METHOD mCallTop : E_cmdState
VAR_INPUT
	I_bExecute		: BOOL;
END_VAR
// No command requested.
IF NOT I_bExecute 
	THEN
    mCallTop       := E_CmdState.Idle;
    RETURN;
END_IF

// Command cylinder to top.
// ToBottom=FALSE, ToTop=TRUE.
fbBottomOut.bBoolValue 		 := FALSE;
fbTopOut.bBoolValue    	   := TRUE;

// Wait until top sensor is active.
IF fbTopIn.bBoolValue 
	THEN
		mCallTop 			 := E_CmdState.Succeeded;
ELSE
    mCallTop 			 := E_CmdState.Busy;
END_IF
END_METHOD

END_FUNCTION_BLOCK

// ---- 1000 Maschine xxx/_Customer/VISUs/Visu_Customer.TcVIS
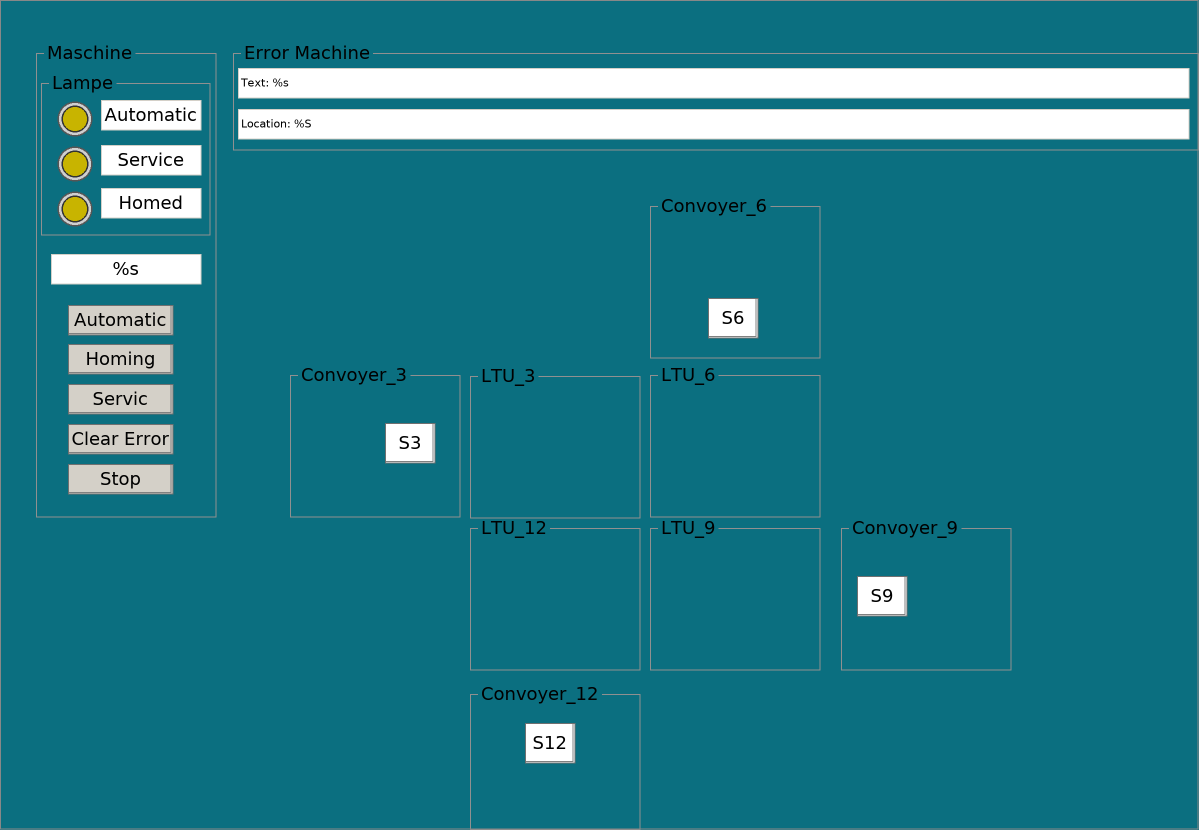
VISUALIZATION Visu_Customer  // 1199x830
    GroupBox (36,45 180x472), "Maschine"
        GroupBox (5,30 169x160), "Lampe"
            Lamp1 (14,114 40x40), variable: MAIN.fbCustomer.stHMI.bHomed, style: Lamp-Lamp1-Yellow
            Lamp1 (14,69 40x40), style: Lamp-Lamp1-Yellow
            Lamp1 (14,24 40x40), style: Lamp-Lamp1-Yellow
            Textfield (60,25 100x30), "Automatic"
            Textfield (60,70 100x30), "Service"
            Textfield (60,113 100x30), "Homed"
        Textfield (15,209 150x30), "%s", text variable: MAIN.fbCustomer.stHMI.eMode
            OnMouseClick: write the text variable via Default
        Button (32,419 105x30), "Stop"
        Button (32,379 105x30), "Clear Error"
        Button (32,339 105x30), "Servic", colour toggle: MAIN.fbCustomer.stHMI.bCmdService
            OnMouseClick: toggle MAIN.fbCustomer.stHMI.bCmdService
        Button (32,299 105x30), "Homing", colour toggle: MAIN.fbCustomer.stHMI.bCmdHome
            OnMouseClick: toggle MAIN.fbCustomer.stHMI.bCmdHome
        Button (32,260 105x30), "Automatic", text variable: MAIN.fbCustomer.stHMI.bCmdAuto, colour toggle: MAIN.fbCustomer.stHMI.bCmdAuto
            OnMouseClick: toggle MAIN.fbCustomer.stHMI.bCmdAuto
    GroupBox (290,367 170x150), "Convoyer_3"
        Button (95,56 50x40), "S3", colour toggle: MAIN.fbCustomer.fdConvoyerDevice3.fbStopperCarrieConvoyer.bHmiSimCarrie
            OnMouseClick: toggle MAIN.fbCustomer.fdConvoyerDevice3.fbStopperCarrieConvoyer.bHmiSimCarrie
    GroupBox (470,368 170x150), "LTU_3"
    GroupBox (650,367 170x150), "LTU_6"
    GroupBox (650,520 170x150), "LTU_9"
    GroupBox (470,520 170x150), "LTU_12"
    GroupBox (650,198 170x160), "Convoyer_6"
        Button (58,100 50x40), "S6", colour toggle: MAIN.fbCustomer.fdConvoyerDevice6.fbStopperCarrieConvoyer.bHmiSimCarrie
            OnMouseClick: toggle MAIN.fbCustomer.fdConvoyerDevice6.fbStopperCarrieConvoyer.bHmiSimCarrie
    GroupBox (470,686 170x144), "Convoyer_12"
        Button (55,37 50x40), "S12", colour toggle: MAIN.fbCustomer.fdConvoyerDevice12.fbStopperCarrieConvoyer.bHmiSimCarrie
            OnMouseClick: toggle MAIN.fbCustomer.fdConvoyerDevice12.fbStopperCarrieConvoyer.bHmiSimCarrie
    GroupBox (841,520 170x150), "Convoyer_9"
        Button (16,56 50x40), "S9", colour toggle: MAIN.fbCustomer.fdConvoyerDevice9.fbStopperCarrieConvoyer.bHmiSimCarrie
            OnMouseClick: toggle MAIN.fbCustomer.fdConvoyerDevice9.fbStopperCarrieConvoyer.bHmiSimCarrie
    GroupBox (233,45 966x105), "Error Machine"
        Textfield (5,23 951x30), "Text: %s"
        Textfield (5,64 951x30), "Location: %S"
END_VISUALIZATION

// ---- GlobalTextList.TcGTLO
TEXTLIST GlobalTextList
  325 = '%s'
  279 = '12'
  584 = 'Auto'
  173 = 'Automatic'
  1066 = 'BASEPOS'
  355 = 'BasePos'
  790 = 'C3'
  669 = 'C6'
  844 = 'Clear Error'
  626 = 'Convoyer_12'
  213 = 'Convoyer_3'
  419 = 'Convoyer_6'
  374 = 'Convoyer_9'
  648 = 'Error'
  908 = 'Error Machine'
  728 = 'Gruppenfeld'
  1008 = 'HOLD'
  917 = 'Homed'
  551 = 'Homing'
  218 = 'Lampe'
  354 = 'Location: %S'
  649 = 'LTU6'
  478 = 'Ltu_12'
  324 = 'LTU_12'
  891 = 'Ltu_3'
  699 = 'LTU_3'
  330 = 'Ltu_6'
  225 = 'LTU_6'
  558 = 'Ltu_9'
  195 = 'LTU_9'
  56 = 'Machine Desk'
  924 = 'Maschine'
  938 = 'Run'
  903 = 'S12'
  136 = 'S3'
  59 = 'S6'
  525 = 'S9'
  585 = 'Semi-Auto'
  238 = 'Servic'
  583 = 'Service'
  85 = 'START'
  779 = 'STOP'
  718 = 'Stop'
  597 = 'Text: %s'
  3265 = 'UI am a live'
END_TEXTLIST
